(* PLC project PRG_ACQUISITION_CFC.project, CODESYS CODESYS V3.5 SP19 Patch 1 *)
(* stored: creationDateTime 2026-08-03T00:00:00, modificationDateTime 2026-08-03T00:00:00 *)

PROGRAM PRG_ACQUISITION_CFC
  VAR
    instAcquisition : FB_AcquisitionLegacyBridge;
  END_VAR
  VAR_OUTPUT
    HwReal : ST_HardwareImage;
    HwSim : ST_HardwareImage;
    HwIn : ST_HardwareImage;
    WinchInputSourceChanged : BOOL;
    TranslationPosTremie : BOOL;
    TranslationPosPV : BOOL;
    TranslationPosP2 : BOOL;
    TranslationPosP1 : BOOL;
    TranslationPosMaintenance : BOOL;
    M3_StatusWord_Filtered : UINT;
    M3_ActualFrequencyHz_Filtered : UINT;
    M3_LimitSwitchFwd : BOOL;
    M3_LimitSwitchRev : BOOL;
    M3_SensorWordIncoherent : BOOL;
    M3_SensorsWord : BYTE;
  END_VAR

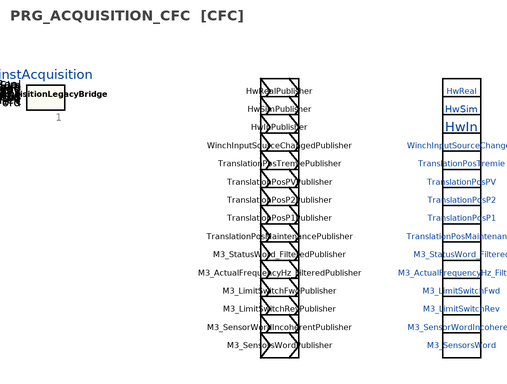
(* CFC diagram, written out as Structured Text *)
instAcquisition();
HwReal := instAcquisition.HwReal;
HwSim := instAcquisition.HwSim;
HwIn := instAcquisition.HwIn;
WinchInputSourceChanged := instAcquisition.WinchInputSourceChanged;
TranslationPosTremie := instAcquisition.TranslationPosTremie;
TranslationPosPV := instAcquisition.TranslationPosPV;
TranslationPosP2 := instAcquisition.TranslationPosP2;
TranslationPosP1 := instAcquisition.TranslationPosP1;
TranslationPosMaintenance := instAcquisition.TranslationPosMaintenance;
M3_StatusWord_Filtered := instAcquisition.M3_StatusWord_Filtered;
M3_ActualFrequencyHz_Filtered := instAcquisition.M3_ActualFrequencyHz_Filtered;
M3_LimitSwitchFwd := instAcquisition.M3_LimitSwitchFwd;
M3_LimitSwitchRev := instAcquisition.M3_LimitSwitchRev;
M3_SensorWordIncoherent := instAcquisition.M3_SensorWordIncoherent;
M3_SensorsWord := instAcquisition.M3_SensorsWord;
END_PROGRAM
